TYPE ST_AutoTuneGains :
STRUCT
	fKp					:LREAL;
	fTn					:LREAL;
	fTv					:LREAL;
	fTd					:LREAL;	
END_STRUCT
END_TYPE

(* stored: Version 1.1.0.1, ProductVersion 3.1.4024.12
   DUT ST_AutoTuneGains: Id {0072efc6-9fc0-4224-8e10-b972663c3c6b} *)
